PROGRAM P_Demo_FB_DALIV2QueryMissingShortAddress
VAR
    fbFB_DALIV2QueryMissingShortAddress        : FB_DALIV2QueryMissingShortAddress;
    stCommandBuffer : ST_DALIV2CommandBuffer;

    bTrigger        : BOOL;
    nLampAddr        : BYTE := 0;

    bResult          : BOOL;

    bBusy           : BOOL;
    bErr            : BOOL;
    nErrId          : UDINT;
END_VAR

// =============================================================================
// 场景：巡检 short addr 0：查询灯具是否丢失短地址（短地址 = MASK）。
//
// 价值：HMI 显示用。
//
// 验证步骤：
//   1. 通信 FB 跑起；编译；登录。
//   2. 在线 bTrigger 一次上升沿；等 bBusy 回 FALSE。
//   3. 观察 fbFB_DALIV2QueryMissingShortAddress.bQueryData 应为预期值（参考本 FB 文档 §4 描述）。
// =============================================================================
fbFB_DALIV2QueryMissingShortAddress(
    bStart           := bTrigger,
    nAddr            := nLampAddr,
    eAddrType        := eDALIV2AddrTypeShort,
    eCommandPriority := eDALIV2CommandPriorityLow,
    stCommandBuffer  := stCommandBuffer
);

bBusy  := fbFB_DALIV2QueryMissingShortAddress.bBusy;
bErr   := fbFB_DALIV2QueryMissingShortAddress.bError;
nErrId := fbFB_DALIV2QueryMissingShortAddress.nErrorId;

END_PROGRAM

(* stored: Version 1.1.0.1, ProductVersion 3.1.4024.5
   POU P_Demo_FB_DALIV2QueryMissingShortAddress: Id {548570b7-3b71-5b62-a58c-873311c41b1f}, SpecialFunc None *)
